// TIA Portal V18 export
FUNCTION "Output_Estop" : Void   // FC31, LAD
{ S7_Optimized_Access := 'TRUE' }
VERSION : 0.1
// stored: AutoNumber true, IsIECCheckEnabled false, SetENOAutomatically false, UDAEnableTagReadback false
   VAR_TEMP
      spare : Bool;
      spare2 : Bool;
      spare3 : Bool;
   END_VAR
BEGIN

REGION Network 1: gear Pump A
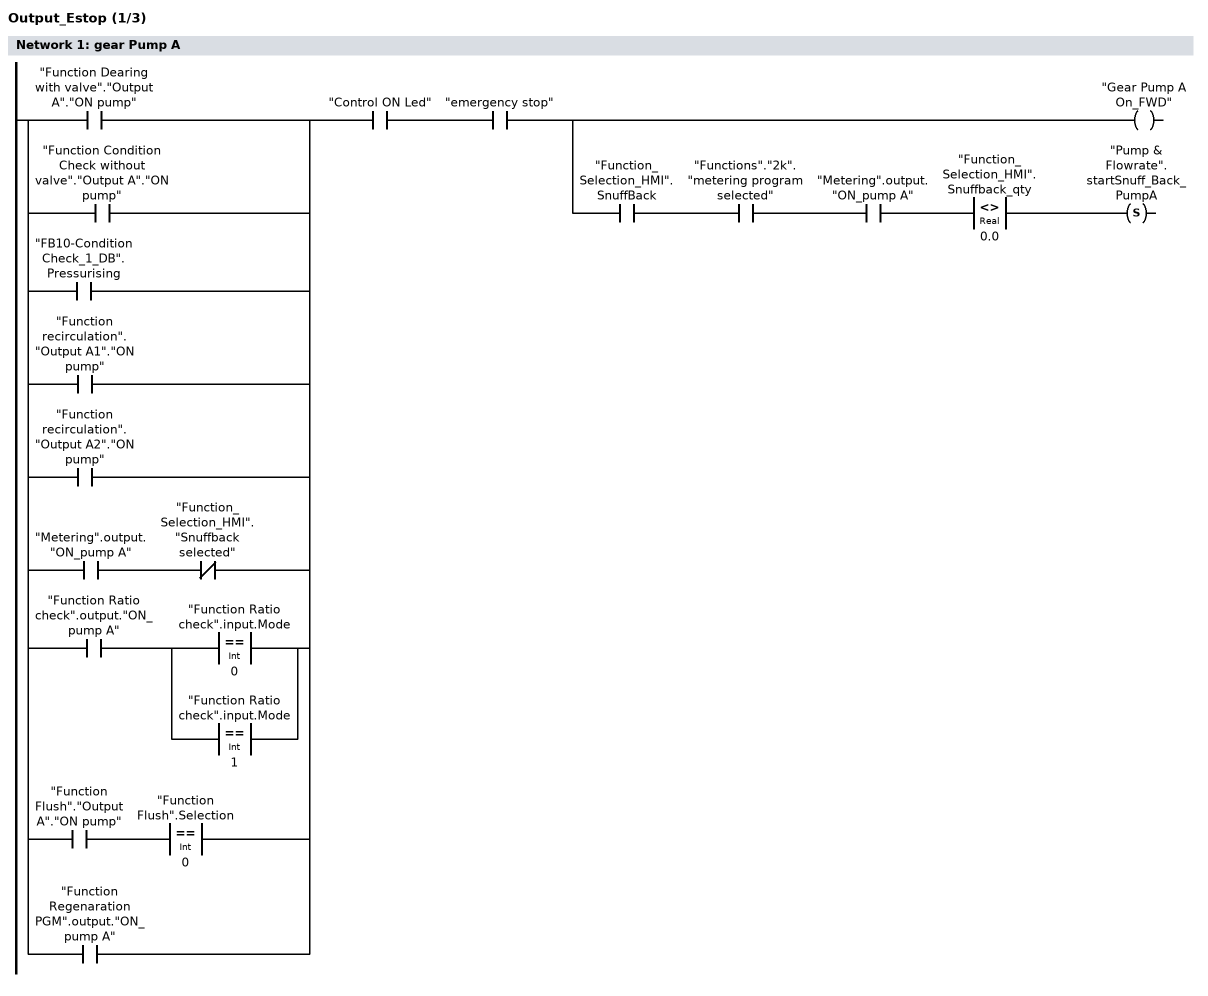
   RUNG wire#powerrail
      Contact( "Function Dearing with valve"."Output A"."ON pump" )
      wire#w1
      Contact( "Control ON Led" )
      Contact( "emergency stop" )
      wire#w3
      Coil( "Gear Pump A On_FWD" )
   END_RUNG
   RUNG wire#powerrail
      Contact( "Function ConditionCheck without valve"."Output A"."ON pump" )
   END_RUNG wire#w1
   RUNG wire#powerrail
      Contact( "FB10-Condition Check_1_DB".Pressurising )
   END_RUNG wire#w1
   RUNG wire#powerrail
      Contact( "Function recirculation"."Output A1"."ON pump" )
   END_RUNG wire#w1
   RUNG wire#powerrail
      Contact( "Function recirculation"."Output A2"."ON pump" )
   END_RUNG wire#w1
   RUNG wire#powerrail
      Contact( "Metering".output."ON_pump A" )
      I_Contact( "Function_Selection_HMI"."Snuffback selected" )
   END_RUNG wire#w1
   RUNG wire#powerrail
      Contact( "Function Ratio check".output."ON_pump A" )
      wire#w2
      { S7_Templates := "SrcType := Int" } EQ_Contact(in1 := "Function Ratio check".input.Mode, in2 := 0)
   END_RUNG wire#w1
   RUNG wire#w2
      { S7_Templates := "SrcType := Int" } EQ_Contact(in1 := "Function Ratio check".input.Mode, in2 := 1)
   END_RUNG wire#w1
   RUNG wire#powerrail
      Contact( "Function Flush"."Output A"."ON pump" )
      { S7_Templates := "SrcType := Int" } EQ_Contact(in1 := "Function Flush".Selection, in2 := 0)
   END_RUNG wire#w1
   RUNG wire#powerrail
      Contact( "Function Regenaration PGM".output."ON_pump A" )
   END_RUNG wire#w1
   RUNG wire#w3
      Contact( "Function_Selection_HMI".SnuffBack )
      Contact( "Functions"."2k"."metering program selected" )
      Contact( "Metering".output."ON_pump A" )
      { S7_Templates := "SrcType := Real" } NE_Contact(in1 := "Function_Selection_HMI".Snuffback_qty, in2 := 0.0)
      S_Coil( "Pump & Flowrate".startSnuff_Back_PumpA )
   END_RUNG
   // the same network as SCL:
   "Gear Pump A On_FWD" := ("Function Dearing with valve"."Output A"."ON pump" OR "Function ConditionCheck without valve"."Output A"."ON pump" OR "FB10-Condition Check_1_DB".Pressurising OR "Function recirculation"."Output A1"."ON pump" OR "Function recirculation"."Output A2"."ON pump" OR ("Metering".output."ON_pump A" AND NOT "Function_Selection_HMI"."Snuffback selected") OR ("Function Ratio check".output."ON_pump A" AND (("Function Ratio check".input.Mode = 0) OR ("Function Ratio check".input.Mode = 1))) OR ("Function Flush"."Output A"."ON pump" AND ("Function Flush".Selection = 0)) OR "Function Regenaration PGM".output."ON_pump A") AND "Control ON Led" AND "emergency stop";
   IF "Gear Pump A On_FWD" AND "Function_Selection_HMI".SnuffBack AND "Functions"."2k"."metering program selected" AND "Metering".output."ON_pump A" AND ("Function_Selection_HMI".Snuffback_qty <> 0.0) THEN
       "Pump & Flowrate".startSnuff_Back_PumpA := TRUE;
   END_IF;
END_REGION

REGION Network 2: gear Pump B
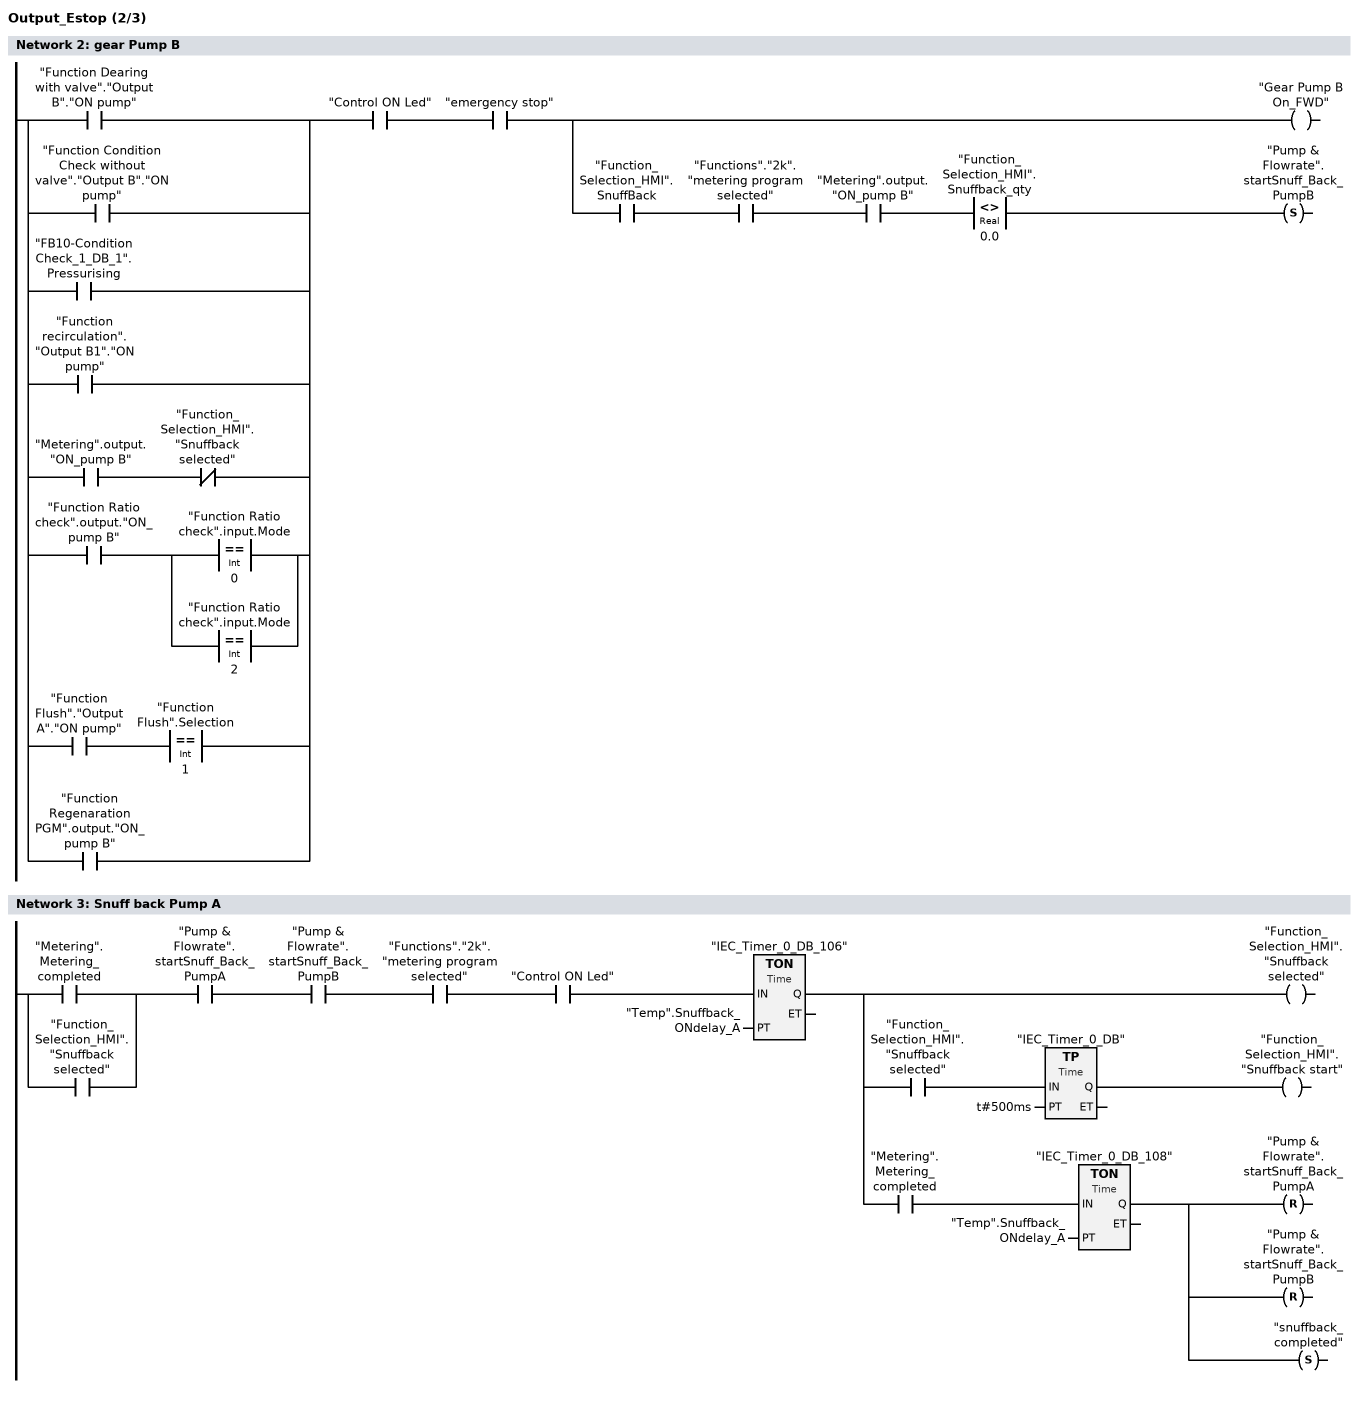
   RUNG wire#powerrail
      Contact( "Function Dearing with valve"."Output B"."ON pump" )
      wire#w1
      Contact( "Control ON Led" )
      Contact( "emergency stop" )
      wire#w3
      Coil( "Gear Pump B On_FWD" )
   END_RUNG
   RUNG wire#powerrail
      Contact( "Function ConditionCheck without valve"."Output B"."ON pump" )
   END_RUNG wire#w1
   RUNG wire#powerrail
      Contact( "FB10-Condition Check_1_DB_1".Pressurising )
   END_RUNG wire#w1
   RUNG wire#powerrail
      Contact( "Function recirculation"."Output B1"."ON pump" )
   END_RUNG wire#w1
   RUNG wire#powerrail
      Contact( "Metering".output."ON_pump B" )
      I_Contact( "Function_Selection_HMI"."Snuffback selected" )
   END_RUNG wire#w1
   RUNG wire#powerrail
      Contact( "Function Ratio check".output."ON_pump B" )
      wire#w2
      { S7_Templates := "SrcType := Int" } EQ_Contact(in1 := "Function Ratio check".input.Mode, in2 := 0)
   END_RUNG wire#w1
   RUNG wire#w2
      { S7_Templates := "SrcType := Int" } EQ_Contact(in1 := "Function Ratio check".input.Mode, in2 := 2)
   END_RUNG wire#w1
   RUNG wire#powerrail
      Contact( "Function Flush"."Output A"."ON pump" )
      { S7_Templates := "SrcType := Int" } EQ_Contact(in1 := "Function Flush".Selection, in2 := 1)
   END_RUNG wire#w1
   RUNG wire#powerrail
      Contact( "Function Regenaration PGM".output."ON_pump B" )
   END_RUNG wire#w1
   RUNG wire#w3
      Contact( "Function_Selection_HMI".SnuffBack )
      Contact( "Functions"."2k"."metering program selected" )
      Contact( "Metering".output."ON_pump B" )
      { S7_Templates := "SrcType := Real" } NE_Contact(in1 := "Function_Selection_HMI".Snuffback_qty, in2 := 0.0)
      S_Coil( "Pump & Flowrate".startSnuff_Back_PumpB )
   END_RUNG
   // the same network as SCL:
   "Gear Pump B On_FWD" := ("Function Dearing with valve"."Output B"."ON pump" OR "Function ConditionCheck without valve"."Output B"."ON pump" OR "FB10-Condition Check_1_DB_1".Pressurising OR "Function recirculation"."Output B1"."ON pump" OR ("Metering".output."ON_pump B" AND NOT "Function_Selection_HMI"."Snuffback selected") OR ("Function Ratio check".output."ON_pump B" AND (("Function Ratio check".input.Mode = 0) OR ("Function Ratio check".input.Mode = 2))) OR ("Function Flush"."Output A"."ON pump" AND ("Function Flush".Selection = 1)) OR "Function Regenaration PGM".output."ON_pump B") AND "Control ON Led" AND "emergency stop";
   IF "Gear Pump B On_FWD" AND "Function_Selection_HMI".SnuffBack AND "Functions"."2k"."metering program selected" AND "Metering".output."ON_pump B" AND ("Function_Selection_HMI".Snuffback_qty <> 0.0) THEN
       "Pump & Flowrate".startSnuff_Back_PumpB := TRUE;
   END_IF;
END_REGION

REGION Network 3: Snuff back Pump A
   RUNG wire#powerrail
      Contact( "Metering".Metering_completed )
      wire#w1
      Contact( "Pump & Flowrate".startSnuff_Back_PumpA )
      Contact( "Pump & Flowrate".startSnuff_Back_PumpB )
      Contact( "Functions"."2k"."metering program selected" )
      Contact( "Control ON Led" )
      { S7_Templates := "time_type := Time" } "IEC_Timer_0_DB_106".TON(pt := "Temp".Snuffback_ONdelay_A, et =>)
      wire#w2
      Coil( "Function_Selection_HMI"."Snuffback selected" )
   END_RUNG
   RUNG wire#powerrail
      Contact( "Function_Selection_HMI"."Snuffback selected" )
   END_RUNG wire#w1
   RUNG wire#w2
      Contact( "Function_Selection_HMI"."Snuffback selected" )
      { S7_Templates := "time_type := Time" } "IEC_Timer_0_DB".TP(pt := t#500ms, et =>)
      Coil( "Function_Selection_HMI"."Snuffback start" )
   END_RUNG
   RUNG wire#w2
      Contact( "Metering".Metering_completed )
      { S7_Templates := "time_type := Time" } "IEC_Timer_0_DB_108".TON(pt := "Temp".Snuffback_ONdelay_A, et =>)
      wire#w3
      R_Coil( "Pump & Flowrate".startSnuff_Back_PumpA )
   END_RUNG
   RUNG wire#w3
      R_Coil( "Pump & Flowrate".startSnuff_Back_PumpB )
   END_RUNG
   RUNG wire#w3
      S_Coil( "snuffback_completed" )
   END_RUNG
   // the same network as SCL:
   "IEC_Timer_0_DB_106".TON(IN := ("Metering".Metering_completed OR "Function_Selection_HMI"."Snuffback selected") AND "Pump & Flowrate".startSnuff_Back_PumpA AND "Pump & Flowrate".startSnuff_Back_PumpB AND "Functions"."2k"."metering program selected" AND "Control ON Led",
                           PT := "Temp".Snuffback_ONdelay_A);
   "Function_Selection_HMI"."Snuffback selected" := "IEC_Timer_0_DB_106".Q;
   "IEC_Timer_0_DB".TP(IN := "IEC_Timer_0_DB_106".Q AND "Function_Selection_HMI"."Snuffback selected",
                       PT := t#500ms);
   "Function_Selection_HMI"."Snuffback start" := "IEC_Timer_0_DB".Q;
   "IEC_Timer_0_DB_108".TON(IN := "IEC_Timer_0_DB_106".Q AND "Metering".Metering_completed,
                           PT := "Temp".Snuffback_ONdelay_A);
   IF "IEC_Timer_0_DB_108".Q THEN
       "Pump & Flowrate".startSnuff_Back_PumpA := FALSE;
       "Pump & Flowrate".startSnuff_Back_PumpB := FALSE;
       "snuffback_completed" := TRUE;
   END_IF;
END_REGION

REGION Network 4
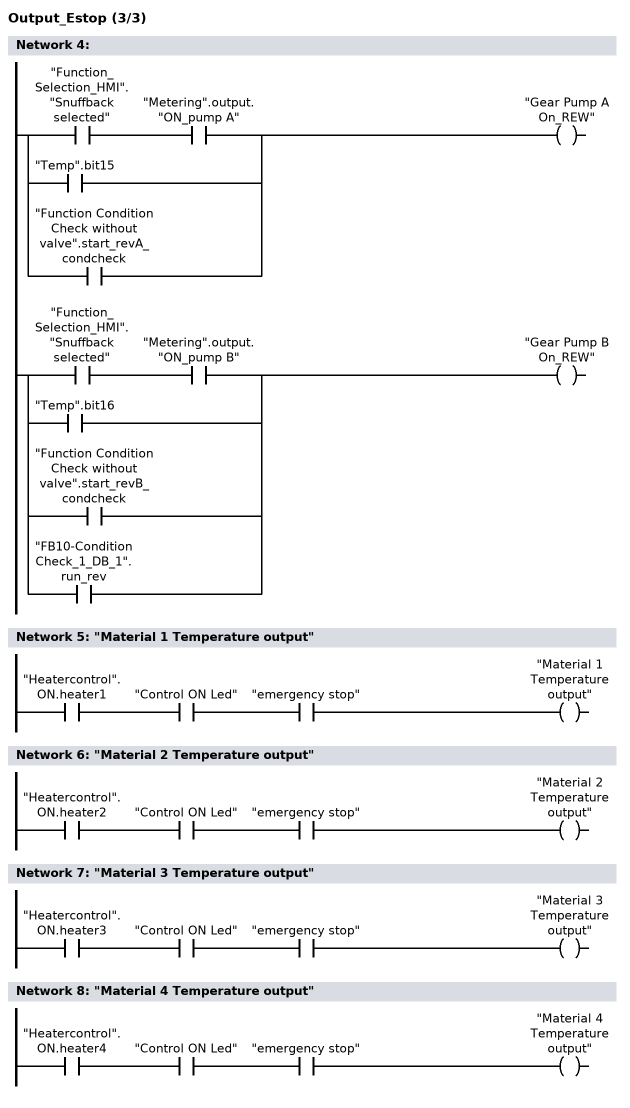
   RUNG wire#powerrail
      Contact( "Function_Selection_HMI"."Snuffback selected" )
      Contact( "Metering".output."ON_pump A" )
      wire#w1
      Coil( "Gear Pump A On_REW" )
   END_RUNG
   RUNG wire#powerrail
      Contact( "Temp".bit15 )
   END_RUNG wire#w1
   RUNG wire#powerrail
      Contact( "Function ConditionCheck without valve".start_revA_condcheck )
   END_RUNG wire#w1
   RUNG wire#powerrail
      Contact( "Function_Selection_HMI"."Snuffback selected" )
      Contact( "Metering".output."ON_pump B" )
      wire#w2
      Coil( "Gear Pump B On_REW" )
   END_RUNG
   RUNG wire#powerrail
      Contact( "Temp".bit16 )
   END_RUNG wire#w2
   RUNG wire#powerrail
      Contact( "Function ConditionCheck without valve".start_revB_condcheck )
   END_RUNG wire#w2
   RUNG wire#powerrail
      Contact( "FB10-Condition Check_1_DB_1".run_rev )
   END_RUNG wire#w2
   // the same network as SCL:
   "Gear Pump A On_REW" := ("Function_Selection_HMI"."Snuffback selected" AND "Metering".output."ON_pump A") OR "Temp".bit15 OR "Function ConditionCheck without valve".start_revA_condcheck;
   "Gear Pump B On_REW" := ("Function_Selection_HMI"."Snuffback selected" AND "Metering".output."ON_pump B") OR "Temp".bit16 OR "Function ConditionCheck without valve".start_revB_condcheck OR "FB10-Condition Check_1_DB_1".run_rev;
END_REGION

REGION Network 5: "Material 1 Temperature output"
   RUNG wire#powerrail
      Contact( "Heatercontrol".ON.heater1 )
      Contact( "Control ON Led" )
      Contact( "emergency stop" )
      Coil( "Material 1 Temperature output" )
   END_RUNG
   // the same network as SCL:
   "Material 1 Temperature output" := "Heatercontrol".ON.heater1 AND "Control ON Led" AND "emergency stop";
END_REGION

REGION Network 6: "Material 2 Temperature output"
   RUNG wire#powerrail
      Contact( "Heatercontrol".ON.heater2 )
      Contact( "Control ON Led" )
      Contact( "emergency stop" )
      Coil( "Material 2 Temperature output" )
   END_RUNG
   // the same network as SCL:
   "Material 2 Temperature output" := "Heatercontrol".ON.heater2 AND "Control ON Led" AND "emergency stop";
END_REGION

REGION Network 7: "Material 3 Temperature output"
   RUNG wire#powerrail
      Contact( "Heatercontrol".ON.heater3 )
      Contact( "Control ON Led" )
      Contact( "emergency stop" )
      Coil( "Material 3 Temperature output" )
   END_RUNG
   // the same network as SCL:
   "Material 3 Temperature output" := "Heatercontrol".ON.heater3 AND "Control ON Led" AND "emergency stop";
END_REGION

REGION Network 8: "Material 4 Temperature output"
   RUNG wire#powerrail
      Contact( "Heatercontrol".ON.heater4 )
      Contact( "Control ON Led" )
      Contact( "emergency stop" )
      Coil( "Material 4 Temperature output" )
   END_RUNG
   // the same network as SCL:
   "Material 4 Temperature output" := "Heatercontrol".ON.heater4 AND "Control ON Led" AND "emergency stop";
END_REGION
END_FUNCTION
